(* Logix 5000 project; controller Prueba2 vendor 1 type 14 code 156 rev 30.11; software revision 30.00 *)

TASK MainTask (continuous, watchdog 500 ms) : MainProgram

MODULES
   Local : vendor 1 type 14 code 156 (Compact 0, rev 30.11)
      DI_4 : 1769-IQ16 (Compact 1, rev 1.1, Input RPI 20 ms)
      DO_5 : vendor 1 type 7 code 86 (Compact 2, rev 2.1, Output RPI 20 ms)
END_MODULES

PROGRAM MainProgram   (* main routine MainRoutine *)
VAR
   A1 : BOOL;
   A2 : BOOL;
   A3 : BOOL;
   A4 : BOOL;
   arranque : BOOL;
   DIstop : ALIAS FOR Local:1:I.Data.0;
   motor1 : BOOL;
   s1 : BOOL;
   s2 : BOOL;
   s3 : BOOL;
   s4 : BOOL;
   salida : BOOL;
   salida1 : BOOL;
   Sensor1 : BOOL := 1;
   Sensor2 : BOOL;
   stop : BOOL;
END_VAR
VAR_INPUT
   start : BOOL;
END_VAR

ROUTINE MainRoutine   (* ladder *)
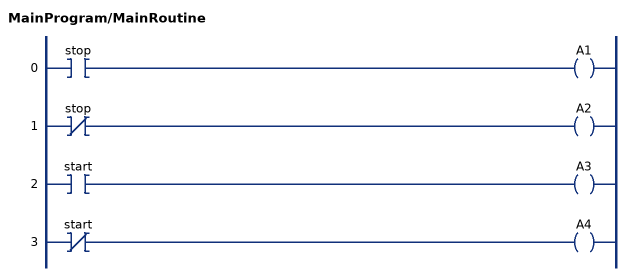
   0: XIC(stop)OTE(A1);
   1: XIO(stop)OTE(A2);
   2: XIC(start)OTE(A3);
   3: XIO(start)OTE(A4);
END_ROUTINE
END_PROGRAM
